// TwinCAT 3 PLC project BMS_Allerstorfer
// ProgramVersion: 3.1.4024.0
// libraries:
//   EfficientIO Communicator, * (EfficientIO)
//   EfficientIO ModbusTCP, * (EfficientIO)
//   Lynus Energy Basic, * (Lynus AG)
//   Lynus Persistent Data V1, * (Lynus AG)
//   Lynus Standards, * (Lynus AG)
//   Tc2_IoFunctions, * (Beckhoff Automation GmbH)
//   Tc2_ModbusSrv, * (Beckhoff Automation GmbH)
//   Tc2_Standard, * (Beckhoff Automation GmbH)
//   Tc2_System, * (Beckhoff Automation GmbH)
//   Tc2_Utilities, * (Beckhoff Automation GmbH)
//   Tc3_BA_Common, * (Beckhoff Automation GmbH)
//   Tc3_Module, * (Beckhoff Automation GmbH)
// project tree:
//   / FastTask.TcTTO, MiddleTask.TcTTO, SlowTask.TcTTO
//   FB/ FB_3HeaterControl.TcPOU, FB_HourCounter.TcPOU, FB_LinearEquation.TcPOU (not stored), FB_PID_T.TcPOU (not stored), FB_RAMP.TcPOU, FB_Symo_PV_Inverter_FLOAT_1_DM_30_InclDisable.TcPOU (not stored), FB_Symo_PV_Inverter_FLOAT_1_DM_30_InclDisable_original.TcPOU
//   POUs/ prgComEffIO.TcPOU, prgEMS.TcPOU, prgGrid.TcPOU, prgHouse.TcPOU, prgPersistent.TcPOU, prgPV.TcPOU, prgRWEffIO.TcPOU (not stored), prgTemperature.TcPOU, prgVarEffIO.TcPOU
// real-time tasks:
//   TASK PlcTask1: cycle T#10ms, priority 21, ADS port 351
//   TASK PlcTask: cycle T#10ms, priority 20, ADS port 350
//   TASK SlowTask: cycle T#10ms, priority 22, ADS port 352
// I/O:
//   DEVICE Gerät 2 (CX-BK)
//     Box 1 (CX-BK)
// variable links:
//   BMS_Allerstorfer/BMS_Allerstorfer Instance <-> Device 2 (CX-BK)/Box 1 (CX-BK)
//     MiddleTask Inputs/prgGrid.fbEM1.fbKL3403.byStateCH1 <-> Term 5 (KL3403)/Channel 1/Status
//     MiddleTask Inputs/prgGrid.fbEM1.fbKL3403.byStateCH2 <-> Term 5 (KL3403)/Channel 2/Status
//     MiddleTask Inputs/prgGrid.fbEM1.fbKL3403.byStateCH3 <-> Term 5 (KL3403)/Channel 3/Status
//     MiddleTask Inputs/prgGrid.fbEM1.fbKL3403.iDataInCH1 <-> Term 5 (KL3403)/Channel 1/Daten Ein
//     MiddleTask Inputs/prgGrid.fbEM1.fbKL3403.iDataInCH2 <-> Term 5 (KL3403)/Channel 2/Daten Ein
//     MiddleTask Inputs/prgGrid.fbEM1.fbKL3403.iDataInCH3 <-> Term 5 (KL3403)/Channel 3/Daten Ein
//     MiddleTask Inputs/prgGrid.fbKBusState.uiKBusState_OUT <-> Inputs/State
//     MiddleTask Inputs/prgTemperature.stInData_{1..4}/iDataIn <-> Term 4 (KL3204)/Channel {1..4}/Daten Ein  (4 links)
//     MiddleTask Inputs/prgTemperature.stInData_{1..4}/iState <-> Term 4 (KL3204)/Channel {1..4}/Status  (4 links)
//     MiddleTask Outputs/prgGrid.fbEM1.fbKL3403.byCntrCH1 <-> Term 5 (KL3403)/Channel 1/Kontrolle
//     MiddleTask Outputs/prgGrid.fbEM1.fbKL3403.byCntrCH2 <-> Term 5 (KL3403)/Channel 2/Kontrolle
//     MiddleTask Outputs/prgGrid.fbEM1.fbKL3403.byCntrCH3 <-> Term 5 (KL3403)/Channel 3/Kontrolle
//     MiddleTask Outputs/prgTemperature.mOut_1 <-> Term 3 (KL2408)/Channel 1/Ausgang
//     MiddleTask Outputs/prgTemperature.mOut_2 <-> Term 3 (KL2408)/Channel 2/Ausgang
//     MiddleTask Outputs/prgTemperature.mOut_3 <-> Term 3 (KL2408)/Channel 3/Ausgang
//     MiddleTask Outputs/prgTemperature.stOutData_{1..4}/iCtrl <-> Term 4 (KL3204)/Channel {1..4}/Kontrolle  (4 links)
//     MiddleTask Outputs/prgTemperature.stOutData_{1..4}/iDataOut <-> Term 4 (KL3204)/Channel {1..4}/Daten Aus  (4 links)
//     SlowTask Outputs/prgTemperature.mOut_{4..8} <-> Term 3 (KL2408)/Channel {4..8}/Ausgang  (5 links)

CONFIGURATION BMS_Allerstorfer
    RESOURCE PLC ON TwinCAT3
        TASK FastTask(INTERVAL := T#10ms, PRIORITY := 21);
        TASK MiddleTask(INTERVAL := T#10ms, PRIORITY := 20);
        TASK SlowTask(INTERVAL := T#10ms, PRIORITY := 22);
        PROGRAM prgVarEffIO WITH FastTask : prgVarEffIO;
        PROGRAM prgRWEffIO WITH FastTask : prgRWEffIO;
        PROGRAM prgComEffIO WITH MiddleTask : prgComEffIO;
        PROGRAM prgEMS WITH MiddleTask : prgEMS;
        PROGRAM prgGrid WITH MiddleTask : prgGrid;
        PROGRAM prgHouse WITH MiddleTask : prgHouse;
        PROGRAM prgPersistent WITH MiddleTask : prgPersistent;
        PROGRAM prgTemperature WITH MiddleTask : prgTemperature;
        PROGRAM prgPV WITH MiddleTask : prgPV;
        PROGRAM prgComEffIO WITH SlowTask : prgComEffIO;
    END_RESOURCE
END_CONFIGURATION

// ---- POUs/prgVarEffIO.TcPOU
PROGRAM prgVarEffIO
VAR
	fbVar		: FB_VarInfo_V3;
END_VAR

fbVar(
	bReadInfo:= , 
	eTMCFile:= eSelectTMCFile.eDontUseTMCFile, 
	eSavePositionTMCFile:= eSavePositionOnPLC.ePostionHardDisk, 
	udiCounterFoundVariables=> , 
	bError=> , 
	bBusy=> , 
	byProgress=> , 
	udiErrorCodeOut=> , 
	eErrorVarInfo_Out=> , 
	sVarWithError=> );
	
fbVar(
	bReadInfo:= , 
	eTMCFile:= eSelectTMCFile.eDontUseTMCFile, 
	eSavePositionTMCFile:= eSavePositionOnPLC.ePostionHardDisk, 
	udiCounterFoundVariables=> , 
	bError=> , 
	bBusy=> , 
	byProgress=> , 
	udiErrorCodeOut=> , 
	eErrorVarInfo_Out=> , 
	sVarWithError=> );
	
fbVar(
	bReadInfo:= , 
	eTMCFile:= eSelectTMCFile.eDontUseTMCFile, 
	eSavePositionTMCFile:= eSavePositionOnPLC.ePostionHardDisk, 
	udiCounterFoundVariables=> , 
	bError=> , 
	bBusy=> , 
	byProgress=> , 
	udiErrorCodeOut=> , 
	eErrorVarInfo_Out=> , 
	sVarWithError=> );

END_PROGRAM

// ---- POUs/prgComEffIO.TcPOU
PROGRAM prgComEffIO
VAR
	fbCom		: FB_MqttCommunicator_V3;
	strAuthKey: STRING(INT#14);
END_VAR

fbCom(
	bConnect:= TRUE, 
	strAuthKey:= 'BMS99299754422', 
	sUserName:= '23fb7b57-8617-4e5d-874b-d9d19721e991', 					// adopt MQTT Username
	sUserPassword:= '60c350ff-dfc0-4bd2-861d-a7d102b328dc', 				// adopt MQTT Password
	eSavePositionCertificate:= eSavePositionOnPLC.ePostionHardDisk, 
	bConnected=> , 
	bError=> , 
	hrErrorCode=> , 
	eConnectionState=> , 
	eErrorMessage_Out=> );
	
	(* old
		strAuthKey:= 'EIO08031879806', 
	sUserName:= 'b37f3835-35ae-441a-9870-02e312a14f46', 					// adopt MQTT Username
	sUserPassword:= '800bfb28-4995-4679-af93-39628385cccf', 				// adopt MQTT Password
*)

END_PROGRAM

// ---- POUs/prgEMS.TcPOU
PROGRAM prgEMS
VAR PERSISTENT
	byMaxDepthOfDischrgEPO		: BYTE;							//{#lynus.ag#()}
	byPrioMinChrgBattSOCInEPO	: BYTE;							//{#lynus.ag#()}
	byResChrgfromGridToBatt		: BYTE;							//{#lynus.ag#()}
	byReserveSOCEPO				: BYTE;							//{#lynus.ag#()}
	uiUpdateTime				: UINT;							//{#lynus.ag#()}
	bEnableEMS					: BOOL;							//{#lynus.ag#()}
	bAllowChrgFromGrid			: BOOL;							//{#lynus.ag#()}
	rMainFuseCSEMS				: REAL;							//{#lynus.ag#()}
	iOperationModeEMS			: INT;							//{#lynus.ag#()}
END_VAR
VAR
	fbEMS						: FB_EMS;
	bIsEnableEMS				: BOOL;							//{#lynus.ag#()}
	bStateAllowChrgFromGrid		: BOOL;							//{#lynus.ag#()}
	bHPActivate					: BOOL;							//{#lynus.ag#()}
	bControllingState			: BOOL;							//{#lynus.ag#()}
	iMessageEMS					: INT;							//{#lynus.ag#()}
	rHeartbeatEMS				: REAL;							//{#lynus.ag#()}
	rErrorWarningEMS			: REAL;							//{#lynus.ag#()}
	rReadyEMS					: REAL;							//{#lynus.ag#()}
	rNewBatteryPowerEMS			: REAL;							//{#lynus.ag#()}
END_VAR

fbEMS.stSetupEMS.bAllowChrgFromGrid := bAllowChrgFromGrid;
	fbEMS.stSetupEMS.byMaxDepthOfDischrgEPO := byMaxDepthOfDischrgEPO;
		fbEMS.stSetupEMS.byPrioMinChrgBattSOCInEPO := byPrioMinChrgBattSOCInEPO;
			fbEMS.stSetupEMS.byResChrgfromGridToBatt := byResChrgfromGridToBatt;
				fbEMS.stSetupEMS.byReserveSOCEPO := byReserveSOCEPO;
					fbEMS.stSetupEMS.rSizeMainFuseCS := rMainFuseCSEMS;
						fbEMS.stSetupEMS.uiUpdateTime := uiUpdateTime;

IF iOperationModeEMS = 0 THEN fbEMS.eOperationMode := E_OperatingMode_EMS.eAllOff;
ELSIF iOperationModeEMS = 1 THEN fbEMS.eOperationMode := E_OperatingMode_EMS.eSelfConsumption;	
ELSIF iOperationModeEMS = 2 THEN fbEMS.eOperationMode := E_OperatingMode_EMS.ePeakLoadCapping;
ELSIF iOperationModeEMS = 3 THEN fbEMS.eOperationMode := E_OperatingMode_EMS.eLoadManagement;			
END_IF

fbEMS(
	bEnable:= bEnableEMS, 
	diNrOfEM_IN_ECS:= , 
	stSetupEMS:= , 
	eOperationMode:= , 
	eSpeedModeBackendController:= E_SpeedModeBackendController_EMS.eSlow, 
	eSpeedModeLocalController:= E_SpeedModeLocalController_EMS.eSlow,
	bActivateHP:= bHPActivate, 
	bControllingState:= TRUE, // bControllingState, 
	rHeartbeat:= rHeartbeatEMS, 
	rErrorWarning:= rErrorWarningEMS, 
	rEnergyOptReady:= rReadyEMS, 
	rNewBattPower:= rNewBatteryPowerEMS, 
	eMessageEMS=> iMessageEMS, 
	bStateEnable=> bIsEnableEMS, 
	bStateAllowChrgFromGrid=> bStateAllowChrgFromGrid, 
	bMissingPowerData=> , 
	bSurplusAvailable=> , 
	byProgress=> , 
	uiState_OUT=> , 
	diNrOfEMS_OUT=> , 
	arrMinPrioReached=> , 
	arrMaxPrioReached=> );

END_PROGRAM

// ---- POUs/prgGrid.TcPOU
PROGRAM prgGrid
VAR PERSISTENT
	rSizeGridConn				: REAL;									//{#lynus.ag#()}
	lrCounterGridCon			: LREAL;							//{#lynus.ag#()}
	lrCounterGridProd			: LREAL;							//{#lynus.ag#()}

END_VAR
VAR
	fbKBusState					: FB_K_Bus_State;
	fbEM1						: FB_EM_Beckhoff_KL3403;
	fbGrid						: FB_Grid_Power;
	fbGridCounter				: FB_EnergyCounter;
	lrPowerGrid					: LREAL;							//{#lynus.ag#()}
	lrPowerEM1_1				: LREAL;							//{#lynus.ag#()}
	lrPowerEM1_2				: LREAL;							//{#lynus.ag#()}
	lrPowerEM1_3				: LREAL;							//{#lynus.ag#()}
	lr_GridVoltageL1N_V			: LREAL;							//{#lynus.ag#()}
	lr_GridVoltageL2N_V			: LREAL;							//{#lynus.ag#()}
	lr_GridVoltageL3N_V			: LREAL;							//{#lynus.ag#()}

	lrReactivePowerGrid			: LREAL;							//{#lynus.ag#()}
	lrApparentPowerGrid			: LREAL;							//{#lynus.ag#()}
	lrPowerGridCons				: LREAL;							//{#lynus.ag#()}
	lrPowerGridProd				: LREAL;							//{#lynus.ag#()}
END_VAR

fbKBusState(	uiKBusState_OUT=> , 
				b_Kbus_notOk=> , 
				word_ErrorCount=> );


fbEM1(
	bEnable:= TRUE, 
	bChannel1Invers:= FALSE,				//Invert power data when transformer are mounted upside down
	bChannel2Invers:= FALSE, 
	bChannel3Invers:= false, 
	uiCurrentTransformerRatioL1:= 250, // 250 / 5 A CTs mounted
	uiCurrentTransformerRatioL2:= 250, 
	uiCurrentTransformerRatioL3:= 250, 
	uiKBusState_IN:= fbKBusState.uiKBusState_OUT, 
	stDataEMPower=> , 
	stDataEMCounter=> , 
	stDataEMPowerRealTime=> , 
	stDataEMCounterRealTime=> , 
	diNrOfEM_OUT=> );

lrPowerGrid := fbEM1.stDataEMPower.lrPowerTotal;
lrCounterGridCon := fbEM1.stDataEMCounter.lrTotalCounterEnergy_Consumption;	
lrCounterGridProd := fbEM1.stDataEMCounter.lrTotalCounterEnergy_Production;	
lrPowerEM1_1 := fbEM1.stDataEMPower.lrPowerL1;
lrPowerEM1_2 := fbEM1.stDataEMPower.lrPowerL2;
lrPowerEM1_3 := fbEM1.stDataEMPower.lrPowerL3;

lrReactivePowerGrid:=fbEM1.stDataEMPower.lrReactivePowerTotal;
lrApparentPowerGrid:=fbEM1.stDataEMPower.lrApparentPowerTotal;

lr_GridVoltageL1N_V:=fbEM1.stDataEMPower.lrVoltageL1N;
lr_GridVoltageL2N_V:=fbEM1.stDataEMPower.lrVoltageL2N;
lr_GridVoltageL3N_V:=fbEM1.stDataEMPower.lrVoltageL3N;


fbGrid(
	bEnable:= TRUE, 
	diNrOfEMS_IN:= prgEMS.fbEMS.diNrOfEMS_OUT, 
	diNrOfEM_IN_Grid:= fbEM1.diNrOfEM_OUT, 
	rSizeGridConn:= rSizeGridConn, 
	stDataGrid=> , 
	diNrOfGrid_OUT=> );
	



// EnergyCounter
fbGridCounter(
	byActiveTariff:= 1, 
	lrPowerInput:= lrPowerGrid, 
	lrTotalCounterEnergy_Consumption=> , 
	lrTotalCounterEnergy_Production=> , 
	lrCounterEnergyT1_Consumption=> , 
	lrCounterEnergyT2_Consumption=> , 
	lrCounterEnergyT1_Production=> , 
	lrCounterEnergyT2_Production=> );

IF fbGridCounter.lrTotalCounterEnergy_Production > lrCounterGridProd THEN  	
		lrCounterGridProd := fbGridCounter.lrTotalCounterEnergy_Production;
END_IF

IF fbGridCounter.lrTotalCounterEnergy_Consumption > lrCounterGridCon THEN  	
	lrCounterGridCon := fbGridCounter.lrTotalCounterEnergy_Consumption;
END_IF

lrPowerGridCons := fbEM1.stDataEMPower.lrPowerConsumption;
lrPowerGridProd := fbEM1.stDataEMPower.lrPowerProduction;

END_PROGRAM

// ---- POUs/prgHouse.TcPOU
PROGRAM prgHouse
VAR
	fbHouse				: FB_HouseC_Power_Virtual;
	bHouseEnabled		: BOOL;						//{#lynus.ag#()}
	lrPowerHouse		: LREAL;					//{#lynus.ag#()}
	lrPowerHouse_Manual	: LREAL;					//{#lynus.ag#()}
	lrPowerHouseUndelayed: LREAL;					//{#lynus.ag#()}
END_VAR
VAR PERSISTENT
	bEnableHouse		: BOOL;						//{#lynus.ag#()}
END_VAR

fbHouse(
	bEnable:= bEnableHouse, 
	diNrOfEMS_IN:= prgEMS.fbEMS.diNrOfEMS_OUT, 
	bSetDefault:= , 
	lrCounterConsumptionSetDefault:= , 
	lrCounterProductionSetDefault:= , 
	stDataHouseC=> , 
	diNrOfHouseC_OUT=> );
	
bHouseEnabled := fbHouse.stDataHouseC.bEnabled;
// lrPowerHouse := fbHouse.stDataHouseC.lrPower; 		// not calculating correctly	
lrPowerHouse_Manual := prgPV.lrPowerPV + prgGrid.lrPowerGrid;

lrPowerHouse:= MAX(0,lrPowerHouse_Manual)- prgTemperature.real_PowerHeater;
lrPowerHouseUndelayed := prgGrid.fbEM1.stDataEMPowerRealTime.lrPowerTotal + prgPV.lrPowerPV - prgTemperature.real_PowerHeater;

END_PROGRAM

// ---- POUs/prgPV.TcPOU
PROGRAM prgPV
VAR PERSISTENT
	lrCounterPV				: LREAL;									//{#lynus.ag#()}
	str_IP_PV_1				: STRING(15):= '10.11.90.100';
	arr_b_EnableWrite			: ARRAY[1..30] OF BOOL;								// Enable write function
	arr_m_DisableInverter		: ARRAY[1..30] OF BOOL;								// disable inverter 
	arr_int_InverterSetpoint	: ARRAY[1..30] OF INT;								// inverter setpoint i[1/100 %] 
	real_MainsSetpointRegulate	: REAL:=-20;							//{#lynus.ag#()}
	real_Factor_Calc: REAL:=110;
	rPValue: REAL := 2;
	udint_IValue: UDINT:=250;
	uditn_DValue: UDINT:=30;
	realMaxGridPower_1: REAL:=-35;
	realMaxGridPower_2: REAL:=-40;
END_VAR
VAR
	fbPV_1					: FB_Symo_PV_Inverter_FLOAT_1_DM_30_InclDisable;
	fbPVCounter				: FB_EnergyCounter;
	lrPowerPV				: LREAL;				//{#lynus.ag#()}
	byErrorWarningPV		: BYTE;					//{#lynus.ag#()}
	
	// extend or reduce amount of PV Inverters
	lrPowerPV_1				: LREAL;				//{#lynus.ag#()}
	lrPowerPV_2				: LREAL;				//{#lynus.ag#()}

	int_SetPointInverter	:INT;					//{#lynus.ag#()}

	real_ActualLoadPercent_PV1: REAL;				//{#lynus.ag#()}
	real_ActualLoadPercent_PV2: REAL;				//{#lynus.ag#()}
	real_RegulatroMaxValue_Calc: REAL;				//{#lynus.ag#()}
	FB_PID_Inverter :FB_PID_T;
	ton_PV_On_Delay_after_Off :ARRAY[1..2]OF Ton;
	
	real_Setpoint_PID_In: REAL;					//{#lynus.ag#()}
	real_RegulatroMaxValue_Limit: REAL;				//{#lynus.ag#()}
		
	i: INT;
END_VAR

// write setpoints to PV array
arr_int_InverterSetpoint[1] := int_SetPointInverter;
arr_int_InverterSetpoint[2] := int_SetPointInverter;

// limit mains regulator setpoint
real_MainsSetpointRegulate := LIMIT(-30,real_MainsSetpointRegulate,0); 
 

fbPV_1.arrUnitID_Inverter[1]:=1;
fbPV_1.arr_b_EnableWrite[1] := arr_b_EnableWrite[1];
fbPV_1.arr_m_DisableInverter[1] := arr_m_DisableInverter[1];
fbPV_1.arr_int_InverterSetpoint[1] := arr_int_InverterSetpoint[1];

fbPV_1.arrUnitID_Inverter[2]:=2;
fbPV_1.arr_b_EnableWrite[2] := arr_b_EnableWrite[2];
fbPV_1.arr_m_DisableInverter[2] := arr_m_DisableInverter[2];
fbPV_1.arr_int_InverterSetpoint[2] := arr_int_InverterSetpoint[2];


fbPV_1.arrUnitID_Inverter[1] :=1;
fbPV_1(
	bEnable				:= TRUE, 
	sIPAdress			:= str_IP_PV_1, 			// modify IP Adress
	arrUnitID_Inverter	:= ,
	arr_b_EnableWrite	:=,
	arr_m_DisableInverter := ,
	arrDataSymo10		=> ,
	stDataEMPower_PV	=> , 
	stDataEMCounter_PV	=> , 
	diNrOfEM_OUT_PV		=> );

lrPowerPV_1 := fbPV_1.arrDataSymo10[1].lrPowerAcInverter;
lrPowerPV_2 := fbPV_1.arrDataSymo10[2].lrPowerAcInverter;




lrPowerPV := lrPowerPV_1 + lrPowerPV_2 ;

// EnergyCounter
fbPVCounter(
	byActiveTariff:= 1, 
	lrPowerInput:= 0 - lrPowerPV, 
	lrTotalCounterEnergy_Consumption=> , 
	lrTotalCounterEnergy_Production=> , 
	lrCounterEnergyT1_Consumption=> , 
	lrCounterEnergyT2_Consumption=> , 
	lrCounterEnergyT1_Production=> , 
	lrCounterEnergyT2_Production=> );
	
IF fbPVCounter.lrTotalCounterEnergy_Production > lrCounterPV THEN  	
	lrCounterPV := fbPVCounter.lrTotalCounterEnergy_Production;
END_IF

// calculate maximum regulator value by looking at the nomal inverter power 
// nominal inverter Values	PV1: 27kW / PV2: 27kW 
real_ActualLoadPercent_PV1 := LREAL_TO_REAL(lrPowerPV_1) / 27*100;
real_ActualLoadPercent_PV2 := LREAL_TO_REAL(lrPowerPV_2) / 27*100;

real_RegulatroMaxValue_Calc := 	MAX(real_ActualLoadPercent_PV1,real_ActualLoadPercent_PV2);
real_RegulatroMaxValue_Calc := LIMIT(1,real_RegulatroMaxValue_Calc,100);
real_RegulatroMaxValue_Limit := LIMIT(0,real_RegulatroMaxValue_Calc*real_Factor_Calc,10000);	// add 20% regualtion margin
FB_PID_Inverter.rMaxValue := real_RegulatroMaxValue_Limit;

// mains parallel operation

FB_PID_Inverter.bEnable := TRUE;
FB_PID_Inverter.rSetpoint := LREAL_TO_REAL(- real_MainsSetpointRegulate); 
int_SetPointInverter := REAL_TO_INT(FB_PID_Inverter.rQController);
FB_PID_Inverter.rActualValue:= LREAL_TO_REAL( -prgGrid.fbEM1.stDataEMPowerRealTime.lrPowerTotal);


FB_PID_Inverter(
	bEnable:= , 
	rSetpoint:= , 
	udiIValue:= udint_IValue, 
	udiDValue:= uditn_DValue, 
	udiDamping:= 0, 
	rPValue:= rPValue, 
	rMaxValue:= , 
	rMinValue:= 100, 
	rNeutralZone:= 1, 
	bDirection:= FALSE, 
	rActualValue:= ,
	rQController=> );
	

real_Setpoint_PID_In := FB_PID_Inverter.rSetpoint;



// disable inverters in case of mains power too big
IF prgGrid.fbEM1.stDataEMPowerRealTime.lrPowerTotal < realMaxGridPower_1 THEN
	arr_m_DisableInverter[1] := TRUE;
ELSIF prgGrid.fbEM1.stDataEMPowerRealTime.lrPowerTotal < realMaxGridPower_2 THEN
	arr_m_DisableInverter[2] := TRUE;
END_IF
IF prgGrid.fbEM1.stDataEMPowerRealTime.lrPowerTotal < -50 THEN
	arr_m_DisableInverter[1] := TRUE;
	arr_m_DisableInverter[2] := TRUE;
END_IF
FOR i:= 1 TO 2 BY 1 DO
	IF arr_m_DisableInverter[i] = TRUE THEN
		ton_PV_On_Delay_after_Off[i].IN := TRUE;
	END_IF
	IF ton_PV_On_Delay_after_Off[i].Q THEN
		ton_PV_On_Delay_after_Off[i].IN := FALSE;
		arr_m_DisableInverter[i] := FALSE;
	END_IF
		
END_FOR
ton_PV_On_Delay_after_Off[1]( PT := T#30S); 	
ton_PV_On_Delay_after_Off[2]( PT := T#60S);

END_PROGRAM

// ---- POUs/prgTemperature.TcPOU
PROGRAM prgTemperature
VAR
	
	fb_Config			: FB_KL320xConfig;
	stInData_1   AT%I*		: ST_KL320xInData;
	stOutData_1  AT%Q*		: ST_KL320xOutData;
	stInData_2   AT%I*		: ST_KL320xInData;
	stOutData_2  AT%Q*		: ST_KL320xOutData;
	stInData_3   AT%I*		: ST_KL320xInData;
	stOutData_3  AT%Q*		: ST_KL320xOutData;
	stInData_4   AT%I*		: ST_KL320xInData;
	stOutData_4  AT%Q*		: ST_KL320xOutData;
	stInData_temp	: ST_KL320xInData;
	stOutData_temp	: ST_KL320xOutData;

	x: INT;
	real_Temp_BoilerOben	:REAL;				//{#lynus.ag#()}
	real_Temp_BoilerUnten	:REAL;				//{#lynus.ag#()}
	mOut_1  AT%Q*		: BOOL;
	mOut_2  AT%Q*		: BOOL;
	mOut_3  AT%Q*		: BOOL;
	mOut_4  AT%Q*		: BOOL;
	mOut_5  AT%Q*		: BOOL;
	mOut_6  AT%Q*		: BOOL;
	mOut_7  AT%Q*		: BOOL;
	mOut_8  AT%Q*		: BOOL;
	fb_heater:FB_3HeaterControl;

	b_Heater1_On: BOOL;							//{#lynus.ag#()}
	b_Heater2_On: BOOL;							//{#lynus.ag#()}
	b_Heater3_On: BOOL;							//{#lynus.ag#()}
	b_Heater1_Manual_On: BOOL;							//{#lynus.ag#()}
	b_Heater2_Manual_On: BOOL;							//{#lynus.ag#()}
	b_Heater3_Manual_On: BOOL;							//{#lynus.ag#()}
	real_StepHeaterControl	: REAL;				//{#lynus.ag#()}
	real_PowerHeater1		: REAL;				//{#lynus.ag#()}
	real_PowerHeater2		: REAL;				//{#lynus.ag#()}
	real_PowerHeater3		: REAL;				//{#lynus.ag#()}
	real_PowerHeater		: REAL;				//{#lynus.ag#()}
END_VAR
VAR PERSISTENT
	real_Boiler_SetPoint	: REAL:=70;				//{#lynus.ag#()}
	b_Enable				: BOOL;					//{#lynus.ag#()}

END_VAR




real_Temp_BoilerUnten :=  INT_TO_REAL(stInData_1.iDataIn)/10;
real_Temp_BoilerOben  :=  INT_TO_REAL(stInData_2.iDataIn)/10;

// heater control
fb_heater(
	m_Enbale:= b_Enable , 
	m_Temperature_high:=  MAX(real_Temp_BoilerOben,real_Temp_BoilerUnten)>95, 
	m_Battery_Discharging := FALSE,
	real_Temperature:=  MAX(real_Temp_BoilerOben,real_Temp_BoilerUnten), 
	real_TemperatureSetPoint:= real_Boiler_SetPoint, 
	real_GridPower := LREAL_TO_REAL(prgGrid.lrPowerGrid), 
	real_BatteryPower := 0,
	real_Size_Step1_kW:= 6, 
	real_Size_Step2_kW:= 6, 
	real_Size_Step3_kW:= 6, 
	m_Step1=> b_Heater1_On, 
	m_Step2=> b_Heater2_On, 
	m_Step3=> b_Heater3_On);
	
mOut_1 := 	b_Heater1_On OR b_Heater1_Manual_On;
mOut_2 := 	b_Heater2_On OR b_Heater2_Manual_On;
mOut_3 := 	b_Heater3_On or b_Heater3_Manual_On;


IF mOut_1 THEN
	real_PowerHeater1 := fb_heater.real_Size_Step1_kW;
ELSE
	real_PowerHeater1 := 0;
END_IF
IF mOut_2 THEN
	real_PowerHeater2 := fb_heater.real_Size_Step2_kW;
ELSE
	real_PowerHeater2 := 0;
END_IF
IF mOut_3 THEN
	real_PowerHeater3 := fb_heater.real_Size_Step3_kW;
ELSE
	real_PowerHeater3 := 0;
END_IF
real_StepHeaterControl := SINT_TO_REAL(fb_heater.sint_Steps_On);

real_PowerHeater := real_PowerHeater1 + real_PowerHeater2 + real_PowerHeater3;
	
CASE x OF 
	0:
		fb_Config.bConfigurate := FALSE;
	1:
		stInData_temp  := stInData_1;
		stOutData_1 	:=stOutData_temp ;
	2:
		stInData_temp  := stInData_2;
		stOutData_2 	:=stOutData_temp ;
	3:
		stInData_temp  := stInData_3;
		stOutData_3 	:=stOutData_temp ;
	4:
		stInData_temp  := stInData_4;
		stOutData_4 	:=stOutData_temp ;
	
END_CASE
// set iSetSensorType = 2 for PT1000
fb_Config(
	bConfigurate:= , 
	bReadConfig:= , 
	iSetSensorType:= , 
	tTimeout:= , 
	bBusy=> , 
	bError=> , 
	iErrorId=> , 
	iState=> , 
	iDataIn=> , 
	iTerminalType=> , 
	iSpecialType=> , 
	iFirmwareVersion=> , 
	sDescription=> , 
	sSensorType=> , 
	bTwoWiredConnection=> , 
	stInData:= stInData_temp , 
	stOutData:= stOutData_temp);

END_PROGRAM

// ---- FB/FB_3HeaterControl.TcPOU
FUNCTION_BLOCK FB_3HeaterControl
VAR_INPUT
	m_Enbale					: BOOL;
	m_Temperature_high			: BOOL;
	m_Battery_Discharging		: BOOL;
	real_Temperature			: REAL;
	real_TemperatureSetPoint	: REAL;
	real_GridPower				: REAL;
	real_BatteryPower			: REAL;
	real_Size_Step1_kW			: REAL;
	real_Size_Step2_kW			: REAL;
	real_Size_Step3_kW			: REAL;
	
	
END_VAR
VAR_OUTPUT
	m_Step1						: BOOL;
	m_Step2						: BOOL;
	m_Step3						: BOOL;
END_VAR
VAR
	fb_HourCounter_Step1		: FB_HourCounter;
	fb_HourCounter_Step2		: FB_HourCounter;
	fb_HourCounter_Step3		: FB_HourCounter;
	r_Trig_allOff				: r_trig;
	real_Hours_Step1			: REAL;
	real_Hours_Step2			: REAL;
	real_Hours_Step3			: REAL;	
	arr_sint_StartOrder			: ARRAY[1..3] OF SINT;
	arr_real_LoadSize			: ARRAY[1..3] OF REAL;
	arr_real_Steps				: ARRAY[1..3] OF REAL;
	
	
	int_state					: INT;
	ton_OnDelay_Steps			: Ton;
	time_OnDelay				: TIME:=T#30S;	
	ton_OffDelay_Steps			: Ton;
	time_OffDelay				: TIME:=T#30S;	
	ton_WaitDelay_Steps			: Ton;
	time_WaitDelay				: TIME:=T#30S;	
	sint_Steps_On				: SINT;
	ton_OffDelay2_Steps			: Ton;
	time_OffDelay2				: TIME:=T#15S;	
END_VAR


CASE int_state OF
	0:	// not enabled
		m_Step1 := FALSE;
		m_Step2 := FALSE;
		m_Step3 := FALSE;
		sint_Steps_On := 0;
		ton_OnDelay_Steps.IN := FALSE;
		ton_OffDelay_Steps.IN := FALSE;
		ton_OffDelay2_Steps.IN := FALSE;
		ton_WaitDelay_Steps.IN := FALSE;
		
		IF 	m_Enbale THEN
			int_state := 10;
		END_IF
	
	10: // check that mains power gets more negative thenn step power + 20%
		IF sint_Steps_On <3 THEN 
			IF real_GridPower + arr_real_LoadSize[sint_Steps_On+1]*1.2 < 0 AND NOT m_Temperature_high AND real_Temperature < (real_TemperatureSetPoint-2) THEN 
				ton_OnDelay_Steps.IN := TRUE;
			ELSE
				ton_OnDelay_Steps.IN := FALSE;
			END_IF
		END_IF
		IF ton_OnDelay_Steps.Q THEN
			ton_OnDelay_Steps.IN := FALSE;
			int_state := 11;
		END_IF
		IF sint_Steps_On <>0 THEN 
			IF real_GridPower > 3 OR  real_Temperature > real_TemperatureSetPoint OR (m_Battery_Discharging AND real_BatteryPower > 5) THEN
 				ton_OffDelay_Steps.IN := TRUE;
			ELSE
				ton_OffDelay_Steps.IN := FALSE;
			END_IF
			IF real_GridPower > 10 THEN
 				ton_OffDelay2_Steps.IN := TRUE;
			ELSE
				ton_OffDelay2_Steps.IN := FALSE;
			END_IF
			
			IF ton_OffDelay_Steps.Q THEN
				ton_OffDelay_Steps.IN := FALSE;
				ton_OffDelay2_Steps.IN := FALSE;
				int_state := 12;
			END_IF
			IF m_Temperature_high AND sint_Steps_On <>0 THEN
				ton_OnDelay_Steps.IN := FALSE;
 				ton_OffDelay_Steps.IN := FALSE;
				ton_OffDelay2_Steps.IN := FALSE;
				int_state := 15;
			END_IF
		END_IF
		
		
	11: // count step one up
		sint_Steps_On := sint_Steps_On+1;
		int_state := 20;
		
	12:// count step one down
		sint_Steps_On := sint_Steps_On-1;
		int_state := 20;
	
	15:// Switch off all steps
		sint_Steps_On := 0;
		int_state := 20;
	
	20: // wait state	
		ton_WaitDelay_Steps.IN := TRUE;
		IF ton_WaitDelay_Steps.Q THEN
			ton_WaitDelay_Steps.IN := FALSE;
			int_state := 10;
		END_IF
END_CASE
ton_OnDelay_Steps(PT := time_OnDelay);
ton_OffDelay_Steps(PT := time_OffDelay);
ton_OffDelay2_Steps(PT := time_OffDelay2);
ton_WaitDelay_Steps(PT := time_WaitDelay);

// if not enabled, force state to 0
IF 	NOT m_Enbale THEN
	int_state := 0;
END_IF

// switch on steps according to sint_Steps_On
CASE sint_Steps_On OF
	0:
		m_Step1 := FALSE;
		m_Step2 := FALSE;
		m_Step3 := FALSE;
		
	1:
		m_Step1 := FALSE;
		m_Step2 := FALSE;
		m_Step3 := FALSE;
		IF arr_sint_StartOrder[1] = 1 THEN 
 			m_Step1 := TRUE;
		ELSIF arr_sint_StartOrder[1] = 2 THEN 
			m_Step2 := TRUE;
		ELSIF arr_sint_StartOrder[1] = 3 THEN 
			m_Step3 := TRUE;
		END_IF
	2:
		m_Step1 := FALSE;
		m_Step2 := FALSE;
		m_Step3 := FALSE;
		IF arr_sint_StartOrder[1] = 1 THEN 
 			m_Step1 := TRUE;
		ELSIF arr_sint_StartOrder[1] = 2 THEN 
			m_Step2 := TRUE;
		ELSIF arr_sint_StartOrder[1] = 3 THEN 
			m_Step3 := TRUE;
		END_IF
		IF arr_sint_StartOrder[2] = 1 THEN 
 			m_Step1 := TRUE;
		ELSIF arr_sint_StartOrder[2] = 2 THEN 
			m_Step2 := TRUE;
		ELSIF arr_sint_StartOrder[2] = 3 THEN 
			m_Step3 := TRUE;
		END_IF
	3:
		m_Step1 := TRUE;
		m_Step2 := TRUE;
		m_Step3 := TRUE;		
END_CASE		
	
// find out which step has the lowest running hours
r_Trig_allOff(CLK := NOT m_Step1 AND NOT m_Step2 AND NOT m_Step3);

IF r_Trig_allOff.Q THEN
	IF real_Hours_Step1 <= real_Hours_Step2 AND real_Hours_Step1<=real_Hours_Step3 THEN
		arr_sint_StartOrder[1] := 1;
		IF real_Hours_Step2 <= real_Hours_Step3 THEN
			arr_sint_StartOrder[2] := 2;
			arr_sint_StartOrder[3] := 3;
		ELSE
			arr_sint_StartOrder[2] := 3;
			arr_sint_StartOrder[3] := 2;
		END_IF
	ELSIF real_Hours_Step2 <= real_Hours_Step1 AND real_Hours_Step2<=real_Hours_Step3 THEN
		arr_sint_StartOrder[1] := 2;
		IF real_Hours_Step1 <= real_Hours_Step3 THEN
			arr_sint_StartOrder[2] := 1;
			arr_sint_StartOrder[3] := 3;
		ELSE
			arr_sint_StartOrder[2] := 3;
			arr_sint_StartOrder[3] := 1;
		END_IF
	ELSIF real_Hours_Step3 <= real_Hours_Step1 AND real_Hours_Step3<=real_Hours_Step2 THEN
		arr_sint_StartOrder[1] := 3;
		IF real_Hours_Step1 <= real_Hours_Step2 THEN
			arr_sint_StartOrder[2] := 1;
			arr_sint_StartOrder[3] := 2;
		ELSE
			arr_sint_StartOrder[2] := 2;
			arr_sint_StartOrder[3] := 1;
		END_IF
	END_IF
	arr_real_Steps[1]	:= real_Size_Step1_kW;
	arr_real_Steps[2]	:= real_Size_Step2_kW;
	arr_real_Steps[3]	:= real_Size_Step3_kW;
	
	arr_real_LoadSize[1] :=   arr_real_Steps[arr_sint_StartOrder[1]];
	arr_real_LoadSize[2] :=   arr_real_Steps[arr_sint_StartOrder[2]];
	arr_real_LoadSize[3] :=   arr_real_Steps[arr_sint_StartOrder[3]];
	
END_IF



// hour counter for each step
fb_HourCounter_Step1(	mCounterON:= m_Step1, 
						realHours=> real_Hours_Step1);
						
fb_HourCounter_Step2(	mCounterON:= m_Step2, 
						realHours=> real_Hours_Step2);
						
fb_HourCounter_Step3(	mCounterON:= m_Step3, 
						realHours=> real_Hours_Step3);

END_FUNCTION_BLOCK

// ---- FB/FB_HourCounter.TcPOU
FUNCTION_BLOCK FB_HourCounter
VAR_INPUT
	mCounterON								: BOOL;
END_VAR
VAR_OUTPUT
	realHours								: REAL;
END_VAR
VAR
	wSecond_old: WORD;
	fbGetSystemTime							: NT_GetTime;																					//Function to read out the windows system time on the local plc
	timGetTime								: TON;																							//Timer to activate the function tho read out the windows system time
END_VAR
VAR PERSISTENT
	udintEngineRunningSeconds				: UDINT;
	realHours_Persistent					: REAL;
END_VAR

IF mCounterON THEN
	IF fbGetSystemTime.TIMESTR.wSecond<>wSecond_old THEN
		udintEngineRunningSeconds:=udintEngineRunningSeconds+1;
	END_IF
END_IF
wSecond_old:=fbGetSystemTime.TIMESTR.wSecond;
realHours:=UDINT_TO_REAL(udintEngineRunningSeconds)/3600;
realHours_Persistent:=realHours;

timGetTime(IN:= NOT timGetTime.Q, PT:= T#1S, Q=> , ET=> );

fbGetSystemTime(
	NETID:= , 
	START:= timGetTime.Q AND NOT fbGetSystemTime.BUSY, 
	TMOUT:= , 
	BUSY=> , 
	ERR=> , 
	ERRID=> , 
	TIMESTR=> );

END_FUNCTION_BLOCK

// ---- POUs/prgPersistent.TcPOU
PROGRAM prgPersistent
VAR
	fbUSV		: FB_WritePersistentData_CX81xx;
	fb_Reboot		: NT_reboot;
	m_Reboot		: BOOL:=FALSE;
	uinit_KbusState: UINT;						//{#lynus.ag#()}
END_VAR

fbUSV(
	eSaveModeData:= eUSVSaveMode.eSaveWhenPowerfail, 
	bLoadPersistentDataOk=> , 
	bPowerFailDetect=> , 
	bError=> , 
	bySaveProcess=> , 
	dwStorageLast24h=> , 
	udiErrorCode=> );
	
	
fb_Reboot(	netid := '',
			delay := 2,
			start := m_Reboot);
	


uinit_KbusState := prgGrid.fbKBusState.uiKBusState_OUT;

END_PROGRAM

// ---- FB/FB_RAMP.TcPOU
FUNCTION_BLOCK FB_RAMP
VAR_INPUT
	realRampInput: REAL;		(* input value *)
	mEnableRamp: BOOL;			(* bit=0:Output=Input, bit=1: Ramp active, mZeroOutout has higher priority *)
	mZeroOutput:BOOL;			(* bit=0 normal operation, bit=1 output zero *)
	realRampSpeed: REAL;		(* speed value/second *)
	realRampSampleTime: REAL; 	(* based on 100ns increments *)
	realEqualize: REAL;
END_VAR
VAR_OUTPUT
	realRampOutput: REAL;		(* output value *)
	mRampSaturised: BOOL;		(* ramp on the end *)
END_VAR

VAR
END_VAR

(* 	24NOV2010:
	- new input variable: equalize value => when intput - output < equalize vale then output = input
*)
IF mEnableRamp AND NOT mZeroOutput THEN
	IF ABS(realRampOutput-realRampInput)<realEqualize THEN
		realRampOutput:=realRampInput; (* direct *)
		mRampSaturised:=TRUE;
	ELSE
		IF realRampOutput<realRampInput THEN (* increment *)
			realRampOutput:=realRampOutput+realRampSpeed*realRampSampleTime; (* realSampleTime in s *)
		END_IF
		IF realRampOutput>realRampInput THEN (* decrement *)
			realRampOutput:=realRampOutput-realRampSpeed*realRampSampleTime; (* realSampleTime in s *)
		END_IF
		mRampSaturised:=FALSE;
	END_IF
ELSE
	IF mZeroOutput THEN
		realRampOutput:=0;
	ELSE
		realRampOutput:=realRampInput; (* direct *)
	END_IF
END_IF

END_FUNCTION_BLOCK

// ---- FB/FB_Symo_PV_Inverter_FLOAT_1_DM_30_InclDisable_original.TcPOU
FUNCTION_BLOCK FB_Symo_PV_Inverter_FLOAT_1_DM_30_InclDisable_original
VAR_INPUT PERSISTENT
	bEnable						: BOOL;												//True = Function is enabled, FALSE = Function is dissabled, no new Data
	sIPAdress					: STRING(15);										//IP Adress from the Inverter
	arrUnitID_Inverter			: ARRAY[1..30] OF BYTE;								//Array with the Unit ID's from each Inverter (Max 30 Inverters) (ID = 1 to 247) (0 = No Inverter)
	arr_b_EnableWrite			: ARRAY[1..30] OF BOOL;								// Enable write function
	arr_m_DisableInverter		: ARRAY[1..30] OF BOOL;								// disable inverter 
	arr_int_InverterSetpoint	: ARRAY[1..30] OF INT;								// inverter setpoint i[1/100 %] 
END_VAR
VAR_OUTPUT
	arrDataSymo10				: ARRAY[1..30] OF ST_Symo_PV_OutData;				//Output structure with Data from Symo 10
	stDataEMPower_PV			: ST_ElectricMeter_Output_Power;					//Output structure with Data from Electric Meter PV (Power Data)
	stDataEMCounter_PV			: ST_ElectricMeter_Output_Counter;					//Output structure with Data from Electric Meter PV (Counter Data)
	diNrOfEM_OUT_PV				: DINT;												//Active Number from the Electric Meter for using on other functions
END_VAR
VAR
	fbElMeter					: FB_ElectricMeter;									//Electric Meter Function 
	fbNumberDevice				: FB_NumberOfDevice;								//Function block to calcualte the number of the Device
	fbConvertEnergyRegister		: FB_CV_WORD_TO_DWORD;								//Convert function
	fbMBRead_FC3				: FB_MBReadRegs;									//Modbus Read Function (FC3)
	fbMBWrite_FC16				: FB_MBWriteRegs;									//Modbus Write Function (FC16)
	timDelay					: TON;												//Timer for Delay between Requests
	timTimeout					: TON;												//Timer for Timeout
	timDissableFunctions		: TON;												//Timer to dissable the Function after Lynus_Standards.Constants_General.tTimeDissableLynusFunctions Days without connection to the Lynus Cloud
	timResetConnectionOnGVL		: TON;												//Timer to try reset the connection Flag on the GVL. (When somebody delete the Connection Function and make only a onlinechange)
	FPEnable					: R_TRIG;											//Internal positive Edge
	FPError_FC_3				: R_TRIG;											//Internal positive Edge
	FPError_FC_16				: R_TRIG;											//Internal positive Edge
	PD_String					: FB_PersistentData_String;							//Function to save persistent data 
	stFloat						: ST_UN_FLOAT_CONVERT_DWORD_REAL;					//Convert the Float Raw Value
	arrBuffer_FC3				: ARRAY[1..47] OF WORD;								//Buffer with Data from FC3
	arrBuffer_FC16				: ARRAY[1..6] OF WORD;								//Buffer with Data from FC16
	arrBuffer_FC16_old			: ARRAY[1..30,1..6] OF WORD;								//Buffer with Data from FC16
	arrUnitID_Inverter_CP		: ARRAY[1..30] OF BYTE;								//Array with unit IDs to compare it when we have a change on the Inputs
	arrCurrentL1				: ARRAY[1..30] OF LREAL;							//Array with the Current from L1 from each Inverter
	arrCurrentL2				: ARRAY[1..30] OF LREAL;							//Array with the Current from L2 from each Inverter
	arrCurrentL3				: ARRAY[1..30] OF LREAL;							//Array with the Current from L3 from each Inverter
	arrVoltageL1L2				: ARRAY[1..30] OF LREAL;							//Array with the Voltage from L1-L2 from each Inverter
	arrVoltageL2L3				: ARRAY[1..30] OF LREAL;							//Array with the Voltage from L2-L3 from each Inverter
	arrVoltageL3L1				: ARRAY[1..30] OF LREAL;							//Array with the Voltage from L3-L1 from each Inverter
	arrVoltageL1N				: ARRAY[1..30] OF LREAL;							//Array with the Voltage from L1-N from each Inverter
	arrVoltageL2N				: ARRAY[1..30] OF LREAL;							//Array with the Voltage from L2-N from each Inverter
	arrVoltageL3N				: ARRAY[1..30] OF LREAL;							//Array with the Voltage from L3-N from each Inverter
	arrACPower					: ARRAY[1..30] OF LREAL;							//Array with the AC Power from each Inverter
	arrFrequency				: ARRAY[1..30] OF LREAL;							//Array with the Frequency from each Inverter
	arrApparentPower			: ARRAY[1..30] OF LREAL;							//Array with the Apparent Power from each Inverter
	arrReactivePower			: ARRAY[1..30] OF LREAL;							//Array with the Reactive Power from each Inverter
	arrProductionEnergy			: ARRAY[1..30] OF LREAL;							//Array with the Production Energy from each Inverter
	arrPD						: ARRAY[1..31] OF FB_PersistentData_Number;			//Function to save persistent data
	bErrorDevice				: BOOL;												//When 1 or more Inverters has a Error, then thsi Flag is true
	byInverterInProgress		: BYTE;												//Shows what Inverter is at the moment in Progress in the State machine to read out the data
	byTotalInverter				: BYTE;												//Summ of total Inverters. (Depends on the unit IDs that are not 0.) 
	byLPForInverter				: BYTE; 											//Variable for Loop to calculate some things for the Inverters
	byWaitInStep				: BYTE;												//Wait in Step before start to clean data on PLC
	iStateGVLData				: INT;												//State machine to handle the data on the GVL
	iStateModbusRead			: INT;												//State variable for Statemachine
	iStateModbusWrite			: INT;												//State variable for Statemachine
	iStateModbus_CP				: INT;												//Compare State variable
	diCounterForGVL				: DINT;												//Counter to clean old data on GVL
	lrCheckValue				: LREAL;											//Internal Value to check the value before convert
	lrCounterEnergyProduction	: LREAL;											//Check counter state before write new one
	iStateModbusError			: INT;											//State variable for Statemachine
	byInverterInProgressWrite	: BYTE;
	ton_Wait_write: Ton;
	x: WORD;
	int_WriteSucessCounter: INT;
END_VAR

// {attribute 'hide_all_locals'}

//Creator : Kai Ebensperger
//Company : Lynus AG
//Date : 28.04.2021
//Version : 1.0.0.0

//With this function its possible to read out values from the Symo 10 PV Inverter from the factory Fronius
//This Function read out the Values from 1 Fronius Datamanager with maximal 30 Inverter.
//The protocol to the Inverter is Modbus TCP
//Versions that are supported : 1.1.5-0
//Attention. To access the registers, an offset of 1 must always be subtracted. Register 40001 would then be on register 40000.
//This Function use the FLOAT Format
//You can query the register data of the individual devices using the Modbus device ID (UnitID).
//Each inverter has its own number stored on the display under "Setup" -> "Datcom"-> "Inverter number".
//Inverter number 00 = Modbus ID 100
//Inverter number 01 = Modbus ID 01
//Inverter number 02 = Modbus ID 02 etc.
//Internal in the GVL this function is 1 PV Plant. We display the summ ov all values from each Inverter

//Changes about AC power
//Date : 29.03.2020
//Version : 1.1.0.0

//Date : 22.12.2022
//Version : 1.2.0.0
// STEFAN: added write to setpoint to inverter


//NOTE for diNr.....Designation => 
//_IN = Here Data come in from other Functions or go out to other functions about the GVL
//_OUT = Here Data go out to other functions about the GVL

(*------------------------------------------------------------------------------------------General Input Part---------------------------------------------------------------------------------------------*)

//Check limitation
FOR byLPForInverter := 1 TO 30 BY 1 DO
	arrUnitID_Inverter[byLPForInverter] := LIMIT(0,arrUnitID_Inverter[byLPForInverter],247);
END_FOR

(*-------------------------------------------------------------Calcualte the number of EM System---------------------------------------------------------------*)

fbNumberDevice(
	diActualNumberOfDevices:= Lynus_Standards.GVL_Energy.stNumberOfDevices.diNumberOfElectricMeters, 
	diMaxNumberOfDevices:= Constants_Energy.diMaxNumberOfElectricMeters, 
	udiCounterOnlineChange:= TwinCAT_SystemInfoVarList._AppInfo.OnlineChangeCnt, 
	bNumberIsCalculatet=> , 
	bFPNumberIsCalculatet=> , 
	bOnlineChange=> , 
	diNumberForThisDevice=> diNrOfEM_OUT_PV, 
	diNumberOfTotalDevices=> );

//Write new Numer on GVL
IF fbNumberDevice.bFPNumberIsCalculatet THEN
	Lynus_Standards.GVL_Energy.stNumberOfDevices.diNumberOfElectricMeters := fbNumberDevice.diNumberOfTotalDevices;	
END_IF 

//Delete old Number on GVL
IF fbNumberDevice.bOnlineChange THEN 
	Lynus_Standards.GVL_Energy.stNumberOfDevices.diNumberOfElectricMeters := diNrOfEM_OUT_PV;	
		iStateGVLData := 1; 
END_IF

(*-------------------------------------------------------------Service from Backend is ready and check the connection to backen for dissabel/enable Function---------------------------------------------------------------*)

//Try to reset the variable for connection on the GVL. When all is normal then the Lynus Mqtt connection function set this variable to true in the next cycle
//When we have no connection to the backend then after Lynus_Standards.Constants_General.tTimeDissableLynusFunctions days the Function is dissabled with all of his functionalities
timResetConnectionOnGVL(IN:= NOT timResetConnectionOnGVL.Q, PT:= T#1H, Q=> , ET=> );
	IF timResetConnectionOnGVL.Q THEN Lynus_Standards.GVL_Communicator.bStateConnectionToEnableFunctions := FALSE; END_IF
		IF NOT Lynus_Standards.GVL_Communicator.bStateConnectionToEnableFunctions THEN timDissableFunctions.IN := TRUE; ELSE timDissableFunctions.IN := FALSE; END_IF  
			timDissableFunctions(IN:= , PT:= Lynus_Standards.Constants_General.tTimeDissableLynusFunctions, Q=> , ET=> );

(*------------------------------------------------------------------------------------------Calcualte the Max Number of Inverters---------------------------------------------------------------------------------------------*)
	
byTotalInverter := 0;
	FOR byLPForInverter := 1 TO 30 BY 1 DO
		IF arrUnitID_Inverter[byLPForInverter] <> 0 THEN byTotalInverter := byTotalInverter + 1; END_IF 
	END_FOR	
	
(*------------------------------------------------------------------------------------------State Machine---------------------------------------------------------------------------------------------*)
	
//Enable
FPEnable(CLK:= bEnable, Q=> );
	IF FPEnable.Q AND iStateModbusRead = 0 AND byTotalInverter > 0 THEN iStateModbusRead := 1; END_IF
		IF NOT bEnable OR timDissableFunctions.Q OR byTotalInverter = 0 OR MEMCMP(ADR(arrUnitID_Inverter),ADR(arrUnitID_Inverter_CP),SIZEOF(arrUnitID_Inverter_CP)) <> 0 THEN iStateModbusRead := 0; END_IF

//Timer for delay
timDelay(IN:= , PT:= T#50MS, Q=> , ET=> );	

//Timer for Timeout in Statemachine
	IF iStateModbusRead = iStateModbus_CP THEN timTimeout.IN := TRUE; ELSE timTimeout.IN := FALSE; END_IF
		IF iStateModbusRead = 0 THEN timTimeout.IN := FALSE; END_IF
timTimeout(IN:= , PT:= T#20S, Q=> , ET=> );	

//Statemachine
CASE iStateModbusRead OF
	
	0://Init Step
		iStateModbus_CP := iStateModbusRead;
			timDelay.IN := FALSE;
		
		FOR byLPForInverter := 1 TO 30 BY 1 DO 
			arrDataSymo10[byLPForInverter].bFunctionIsActive := FALSE;
				arrDataSymo10[byLPForInverter].eOperatingStateInverter := E_Symo_PV_OperatingState.eNoDataReceived;
					arrDataSymo10[byLPForInverter].lrPowerAcInverter := 0;
			arrCurrentL1[byLPForInverter] := 0;
				arrCurrentL2[byLPForInverter] := 0;
			arrCurrentL3[byLPForInverter] := 0;
				arrVoltageL1L2[byLPForInverter] := 0;
			arrVoltageL2L3[byLPForInverter] := 0;
				arrVoltageL3L1[byLPForInverter] := 0;
			arrVoltageL1N[byLPForInverter] := 0;
				arrVoltageL2N[byLPForInverter] := 0;
			arrVoltageL3N[byLPForInverter] := 0;
				arrACPower[byLPForInverter] := 0;
			arrFrequency[byLPForInverter] := 0;
				arrApparentPower[byLPForInverter] := 0;
			arrReactivePower[byLPForInverter] := 0;
				arrProductionEnergy[byLPForInverter] := 0;
		END_FOR
				fbMBRead_FC3.bExecute := FALSE;
					lrCheckValue := 0;
			
		//After reset the Arrays when we have a change on the Unit ID's we restart the State Machine
		IF MEMCMP(ADR(arrUnitID_Inverter),ADR(arrUnitID_Inverter_CP),SIZEOF(arrUnitID_Inverter_CP)) <> 0 AND bEnable AND byTotalInverter > 0 THEN
			iStateModbusRead := 1;
				arrUnitID_Inverter_CP := arrUnitID_Inverter;
		END_IF
		
	1://Search the Unit ID to read out the Data for each Inverter with Unit ID <> 0
		iStateModbus_CP := iStateModbusRead;
		
		IF byInverterInProgress >= 30 THEN byInverterInProgress := 0; END_IF
		
		byInverterInProgress := byInverterInProgress + 1;
			byInverterInProgress := LIMIT(1,byInverterInProgress,30);	
		
		IF arrUnitID_Inverter[byInverterInProgress] <> 0 THEN iStateModbusRead := 2; END_IF
				
	2://Read out first Registers from 40072 to 40118
		arrDataSymo10[byInverterInProgress].bFunctionIsActive := TRUE;
			iStateModbus_CP := iStateModbusRead;
		
		fbMBRead_FC3.nQuantity := 47;
			fbMBRead_FC3.nMBAddr := 40071;
				fbMBRead_FC3.bExecute := TRUE;
					fbMBRead_FC3.nUnitID := arrUnitID_Inverter[byInverterInProgress];
			
		IF fbMBRead_FC3.bBusy THEN timDelay.IN := TRUE; END_IF
		
		//Wait for Delay, copy Data and then next step
		IF NOT fbMBRead_FC3.bBusy AND NOT fbMBRead_FC3.bError AND timDelay.Q THEN
			//Copy Data Current L1
			fbConvertEnergyRegister(wInputValue_1:= arrBuffer_FC3[3], wInputValue_2:= arrBuffer_FC3[4], eByteOrderForConvert:= eByteOrder.eBigEndian, dwOutputValue=> );
				stFloat.dwRawValue := fbConvertEnergyRegister.dwOutputValue;
					lrCheckValue := stFloat.rValueFloat;	
						IF lrCheckValue >= - 3.402823E+38 AND lrCheckValue <= 3.402823E+38 THEN 
							arrCurrentL1[byInverterInProgress] := lrCheckValue;
						ELSE
							iStateModbusRead := 300;
								arrDataSymo10[byInverterInProgress].eErrorState := E_Symo_PV_Error.eSymo10TooBigValueReceived;		
						END_IF
			//Copy Data Current L2
			fbConvertEnergyRegister(wInputValue_1:= arrBuffer_FC3[5], wInputValue_2:= arrBuffer_FC3[6], eByteOrderForConvert:= eByteOrder.eBigEndian, dwOutputValue=> );
				stFloat.dwRawValue := fbConvertEnergyRegister.dwOutputValue;
					lrCheckValue := stFloat.rValueFloat;	
						IF lrCheckValue >= - 3.402823E+38 AND lrCheckValue <= 3.402823E+38 THEN 
							arrCurrentL2[byInverterInProgress] := lrCheckValue;
						ELSE
							iStateModbusRead := 300;
								arrDataSymo10[byInverterInProgress].eErrorState := E_Symo_PV_Error.eSymo10TooBigValueReceived;		
						END_IF
			//Copy Data Current L3
			fbConvertEnergyRegister(wInputValue_1:= arrBuffer_FC3[7], wInputValue_2:= arrBuffer_FC3[8], eByteOrderForConvert:= eByteOrder.eBigEndian, dwOutputValue=> );
				stFloat.dwRawValue := fbConvertEnergyRegister.dwOutputValue;
					lrCheckValue := stFloat.rValueFloat;	
						IF lrCheckValue >= - 3.402823E+38 AND lrCheckValue <= 3.402823E+38 THEN 
							arrCurrentL3[byInverterInProgress] := lrCheckValue;
						ELSE
							iStateModbusRead := 300;
								arrDataSymo10[byInverterInProgress].eErrorState := E_Symo_PV_Error.eSymo10TooBigValueReceived;		
						END_IF
			//Copy Data Voltage L1-L2
			fbConvertEnergyRegister(wInputValue_1:= arrBuffer_FC3[9], wInputValue_2:= arrBuffer_FC3[10], eByteOrderForConvert:= eByteOrder.eBigEndian, dwOutputValue=> );
				stFloat.dwRawValue := fbConvertEnergyRegister.dwOutputValue;
					lrCheckValue := stFloat.rValueFloat;	
						IF lrCheckValue >= - 3.402823E+38 AND lrCheckValue <= 3.402823E+38 THEN 
							arrVoltageL1L2[byInverterInProgress] := lrCheckValue;
						ELSE
							iStateModbusRead := 300;
								arrDataSymo10[byInverterInProgress].eErrorState := E_Symo_PV_Error.eSymo10TooBigValueReceived;		
						END_IF
			//Copy Data Voltage L2-L3
			fbConvertEnergyRegister(wInputValue_1:= arrBuffer_FC3[11], wInputValue_2:= arrBuffer_FC3[12], eByteOrderForConvert:= eByteOrder.eBigEndian, dwOutputValue=> );
				stFloat.dwRawValue := fbConvertEnergyRegister.dwOutputValue;
					lrCheckValue := stFloat.rValueFloat;	
						IF lrCheckValue >= - 3.402823E+38 AND lrCheckValue <= 3.402823E+38 THEN 
							arrVoltageL2L3[byInverterInProgress] := lrCheckValue;
						ELSE
							iStateModbusRead := 300;
								arrDataSymo10[byInverterInProgress].eErrorState := E_Symo_PV_Error.eSymo10TooBigValueReceived;		
						END_IF
			//Copy Data Voltage L3-L1
			fbConvertEnergyRegister(wInputValue_1:= arrBuffer_FC3[13], wInputValue_2:= arrBuffer_FC3[14], eByteOrderForConvert:= eByteOrder.eBigEndian, dwOutputValue=> );
				stFloat.dwRawValue := fbConvertEnergyRegister.dwOutputValue;
					lrCheckValue := stFloat.rValueFloat;	
						IF lrCheckValue >= - 3.402823E+38 AND lrCheckValue <= 3.402823E+38 THEN 
							arrVoltageL3L1[byInverterInProgress] := lrCheckValue;
						ELSE
							iStateModbusRead := 300;
								arrDataSymo10[byInverterInProgress].eErrorState := E_Symo_PV_Error.eSymo10TooBigValueReceived;		
						END_IF
			//Copy Data Voltage L1-N
			fbConvertEnergyRegister(wInputValue_1:= arrBuffer_FC3[15], wInputValue_2:= arrBuffer_FC3[16], eByteOrderForConvert:= eByteOrder.eBigEndian, dwOutputValue=> );
				stFloat.dwRawValue := fbConvertEnergyRegister.dwOutputValue;
					lrCheckValue := stFloat.rValueFloat;	
						IF lrCheckValue >= - 3.402823E+38 AND lrCheckValue <= 3.402823E+38 THEN 
							arrVoltageL1N[byInverterInProgress] := lrCheckValue;
						ELSE
							iStateModbusRead := 300;
								arrDataSymo10[byInverterInProgress].eErrorState := E_Symo_PV_Error.eSymo10TooBigValueReceived;		
						END_IF
			//Copy Data Voltage L2-N
			fbConvertEnergyRegister(wInputValue_1:= arrBuffer_FC3[17], wInputValue_2:= arrBuffer_FC3[18], eByteOrderForConvert:= eByteOrder.eBigEndian, dwOutputValue=> );
				stFloat.dwRawValue := fbConvertEnergyRegister.dwOutputValue;
					lrCheckValue := stFloat.rValueFloat;	
						IF lrCheckValue >= - 3.402823E+38 AND lrCheckValue <= 3.402823E+38 THEN 
							arrVoltageL2N[byInverterInProgress] := lrCheckValue;
						ELSE
							iStateModbusRead := 300;
								arrDataSymo10[byInverterInProgress].eErrorState := E_Symo_PV_Error.eSymo10TooBigValueReceived;		
						END_IF
			//Copy Data Voltage L3-N
			fbConvertEnergyRegister(wInputValue_1:= arrBuffer_FC3[19], wInputValue_2:= arrBuffer_FC3[20], eByteOrderForConvert:= eByteOrder.eBigEndian, dwOutputValue=> );
				stFloat.dwRawValue := fbConvertEnergyRegister.dwOutputValue;
					lrCheckValue := stFloat.rValueFloat;	
						IF lrCheckValue >= - 3.402823E+38 AND lrCheckValue <= 3.402823E+38 THEN 
							arrVoltageL3N[byInverterInProgress] := lrCheckValue;
						ELSE
							iStateModbusRead := 300;
								arrDataSymo10[byInverterInProgress].eErrorState := E_Symo_PV_Error.eSymo10TooBigValueReceived;		
						END_IF
			//Copy Data AC Power
			fbConvertEnergyRegister(wInputValue_1:= arrBuffer_FC3[21], wInputValue_2:= arrBuffer_FC3[22], eByteOrderForConvert:= eByteOrder.eBigEndian, dwOutputValue=> );
				stFloat.dwRawValue := fbConvertEnergyRegister.dwOutputValue;
					lrCheckValue := stFloat.rValueFloat;	
						IF lrCheckValue >= - 3.402823E+38 AND lrCheckValue <= 3.402823E+38 THEN 
							arrACPower[byInverterInProgress] := lrCheckValue;
								arrDataSymo10[byInverterInProgress].lrPowerAcInverter := arrACPower[byInverterInProgress] / 1000;
						ELSE
							iStateModbusRead := 300;
								arrDataSymo10[byInverterInProgress].eErrorState := E_Symo_PV_Error.eSymo10TooBigValueReceived;		
						END_IF
			//Copy Data Frequency
			fbConvertEnergyRegister(wInputValue_1:= arrBuffer_FC3[23], wInputValue_2:= arrBuffer_FC3[24], eByteOrderForConvert:= eByteOrder.eBigEndian, dwOutputValue=> );
				stFloat.dwRawValue := fbConvertEnergyRegister.dwOutputValue;
					lrCheckValue := stFloat.rValueFloat;	
						IF lrCheckValue >= - 3.402823E+38 AND lrCheckValue <= 3.402823E+38 THEN 
							arrFrequency[byInverterInProgress] := lrCheckValue;
						ELSE
							iStateModbusRead := 300;
								arrDataSymo10[byInverterInProgress].eErrorState := E_Symo_PV_Error.eSymo10TooBigValueReceived;		
						END_IF
			//Copy Data Apparent Power
			fbConvertEnergyRegister(wInputValue_1:= arrBuffer_FC3[25], wInputValue_2:= arrBuffer_FC3[26], eByteOrderForConvert:= eByteOrder.eBigEndian, dwOutputValue=> );
				stFloat.dwRawValue := fbConvertEnergyRegister.dwOutputValue;
					lrCheckValue := stFloat.rValueFloat;	
						IF lrCheckValue >= - 3.402823E+38 AND lrCheckValue <= 3.402823E+38 THEN 
							arrApparentPower[byInverterInProgress] := lrCheckValue;
						ELSE
							iStateModbusRead := 300;
								arrDataSymo10[byInverterInProgress].eErrorState := E_Symo_PV_Error.eSymo10TooBigValueReceived;		
						END_IF
			//Copy Data Reactive Power
			fbConvertEnergyRegister(wInputValue_1:= arrBuffer_FC3[27], wInputValue_2:= arrBuffer_FC3[28], eByteOrderForConvert:= eByteOrder.eBigEndian, dwOutputValue=> );
				stFloat.dwRawValue := fbConvertEnergyRegister.dwOutputValue;
					lrCheckValue := stFloat.rValueFloat;	
						IF lrCheckValue >= - 3.402823E+38 AND lrCheckValue <= 3.402823E+38 THEN 
							arrReactivePower[byInverterInProgress] := lrCheckValue;
						ELSE
							iStateModbusRead := 300;
								arrDataSymo10[byInverterInProgress].eErrorState := E_Symo_PV_Error.eSymo10TooBigValueReceived;		
						END_IF
			//Copy Data AC production Energy
			fbConvertEnergyRegister(wInputValue_1:= arrBuffer_FC3[31], wInputValue_2:= arrBuffer_FC3[32], eByteOrderForConvert:= eByteOrder.eBigEndian, dwOutputValue=> );
				stFloat.dwRawValue := fbConvertEnergyRegister.dwOutputValue;
					lrCheckValue := stFloat.rValueFloat;	
						IF lrCheckValue >= - 3.402823E+38 AND lrCheckValue <= 3.402823E+38 THEN 
							arrProductionEnergy[byInverterInProgress] := lrCheckValue / 1000;
						ELSE
							iStateModbusRead := 300;
								arrDataSymo10[byInverterInProgress].eErrorState := E_Symo_PV_Error.eSymo10TooBigValueReceived;		
						END_IF
			//Operating State		
			IF arrBuffer_FC3[47] = 1 THEN arrDataSymo10[byInverterInProgress].eOperatingStateInverter := E_Symo_PV_OperatingState.eOff;
				ELSIF arrBuffer_FC3[47] = 2 THEN arrDataSymo10[byInverterInProgress].eOperatingStateInverter := E_Symo_PV_OperatingState.eSleeping;
				ELSIF arrBuffer_FC3[47] = 3 THEN arrDataSymo10[byInverterInProgress].eOperatingStateInverter := E_Symo_PV_OperatingState.eStartingUp;
				ELSIF arrBuffer_FC3[47] = 4 THEN arrDataSymo10[byInverterInProgress].eOperatingStateInverter := E_Symo_PV_OperatingState.eTrackingPowerPoint;
				ELSIF arrBuffer_FC3[47] = 5 THEN arrDataSymo10[byInverterInProgress].eOperatingStateInverter := E_Symo_PV_OperatingState.eForcedPowerReduction;
				ELSIF arrBuffer_FC3[47] = 6 THEN arrDataSymo10[byInverterInProgress].eOperatingStateInverter := E_Symo_PV_OperatingState.eShuttingDown;
				ELSIF arrBuffer_FC3[47] = 7 THEN arrDataSymo10[byInverterInProgress].eOperatingStateInverter := E_Symo_PV_OperatingState.eFaults;
				ELSIF arrBuffer_FC3[47] = 8 THEN arrDataSymo10[byInverterInProgress].eOperatingStateInverter := E_Symo_PV_OperatingState.eStandby;
				ELSE arrDataSymo10[byInverterInProgress].eOperatingStateInverter := E_Symo_PV_OperatingState.eNoDataReceived;
			END_IF
			//Next Step
			IF iStateModbusRead = 2 THEN
				fbMBRead_FC3.bExecute := FALSE;
					timDelay.IN := FALSE;
						iStateModbusRead := 3;
							arrDataSymo10[byInverterInProgress].bError := FALSE; 
								arrDataSymo10[byInverterInProgress].eErrorState := E_Symo_PV_Error.eNoError;
			END_IF
		END_IF
			
		//Error from Inverter
		IF NOT fbMBRead_FC3.bBusy AND NOT fbMBRead_FC3.bError AND timDelay.Q AND arrDataSymo10[byInverterInProgress].eOperatingStateInverter = E_Symo_PV_OperatingState.eFaults THEN
			iStateModbusRead := 300;
				arrDataSymo10[byInverterInProgress].eErrorState := E_Symo_PV_Error.eSymo10Error;
		END_IF
	 
		//Error or Timeout
		IF FPError_FC_3.Q OR timTimeout.Q THEN
			iStateModbusRead := 300;
				arrDataSymo10[byInverterInProgress].eErrorState := E_Symo_PV_Error.eModbusTCPError;
		END_IF

	3://Calculate the sum of the values
		iStateModbus_CP := iStateModbusRead;
		
		lrCounterEnergyProduction := 0;
			fbElMeter.lrCurrentL1 := 0;
		fbElMeter.lrCurrentL2 := 0;	
			fbElMeter.lrCurrentL3 := 0;
		fbElMeter.lrVoltageL1N := 0;
			fbElMeter.lrVoltageL2N := 0;
		fbElMeter.lrVoltageL3N := 0;
			fbElMeter.lrVoltageL1L2 := 0;
		fbElMeter.lrVoltageL2L3 := 0;
			fbElMeter.lrVoltageL3L1 := 0;
		fbElMeter.lrPowerTotal := 0;
			fbElMeter.lrFrequency := 0;
		fbElMeter.lrReactivePowerTotal := 0;
			fbElMeter.lrApparentPowerTotal := 0;
		
		FOR byLPForInverter := 1 TO 30 BY 1 DO 
			lrCounterEnergyProduction := lrCounterEnergyProduction + arrProductionEnergy[byLPForInverter];
			IF lrCounterEnergyProduction > fbElMeter.lrCounterEnergyT1_Production THEN
				fbElMeter.lrCounterEnergyT1_Production := lrCounterEnergyProduction;
			END_IF
				fbElMeter.lrCurrentL1 := fbElMeter.lrCurrentL1 + arrCurrentL1[byLPForInverter];
			fbElMeter.lrCurrentL2 := fbElMeter.lrCurrentL2 + arrCurrentL2[byLPForInverter];	
				fbElMeter.lrCurrentL3 := fbElMeter.lrCurrentL3 + arrCurrentL3[byLPForInverter];
			IF byTotalInverter > 0 THEN
				fbElMeter.lrVoltageL1N := (fbElMeter.lrVoltageL1N + arrVoltageL1N[byLPForInverter]) / byTotalInverter;
					fbElMeter.lrVoltageL2N := (fbElMeter.lrVoltageL2N + arrVoltageL2N[byLPForInverter]) / byTotalInverter;
				fbElMeter.lrVoltageL3N := (fbElMeter.lrVoltageL3N + arrVoltageL3N[byLPForInverter]) / byTotalInverter;
					fbElMeter.lrVoltageL1L2 := (fbElMeter.lrVoltageL1L2 + arrVoltageL1L2[byLPForInverter]) / byTotalInverter;
				fbElMeter.lrVoltageL2L3 := (fbElMeter.lrVoltageL2L3 + arrVoltageL2L3[byLPForInverter]) / byTotalInverter;
					fbElMeter.lrVoltageL3L1 := (fbElMeter.lrVoltageL3L1 + arrVoltageL3L1[byLPForInverter]) / byTotalInverter;
				fbElMeter.lrFrequency := (fbElMeter.lrFrequency + arrFrequency[byLPForInverter]) / byTotalInverter;
			END_IF
					fbElMeter.lrPowerTotal := fbElMeter.lrPowerTotal + arrACPower[byLPForInverter];
				fbElMeter.lrReactivePowerTotal := fbElMeter.lrReactivePowerTotal + arrReactivePower[byLPForInverter];
					fbElMeter.lrApparentPowerTotal := fbElMeter.lrApparentPowerTotal + arrApparentPower[byLPForInverter];
		END_FOR	
					
		fbElMeter.lrTotalCounterEnergy_Production := fbElMeter.lrCounterEnergyT1_Production; 
		
			iStateModbusRead := 4;
	
	4://Wait and go to write
		iStateModbus_CP := iStateModbusRead;
		
		iStateModbusWrite := 1;
		iStateModbusRead := - 1;	
				
	300://Error
		iStateModbus_CP := iStateModbusRead;
		timDelay.IN := FALSE;
		fbMBRead_FC3.bExecute := FALSE;
		arrDataSymo10[byInverterInProgress].bError := TRUE;
		iStateModbusWrite := 1;
		iStateModbusRead := - 1;	
END_CASE
(*------------------------------------------------------------------------------------------State Machine Write---------------------------------------------------------------------------------------------*)	
	
CASE iStateModbusWrite OF	
	1://Search the Unit ID to read out the Data for each Inverter with Unit ID <> 0
		iStateModbus_CP := iStateModbusWrite;
		arr_int_InverterSetpoint[byInverterInProgressWrite] := LIMIT (0,arr_int_InverterSetpoint[byInverterInProgressWrite],10000);
		IF byInverterInProgressWrite >= 30 THEN byInverterInProgressWrite := 0; END_IF
		
		byInverterInProgressWrite := byInverterInProgressWrite + 1;
		byInverterInProgressWrite := LIMIT(1,byInverterInProgressWrite,30);	
		
		IF arrUnitID_Inverter[byInverterInProgressWrite] <> 0 THEN iStateModbusWrite := 2; END_IF
				

	2://write disable inverter bit
		iStateModbus_CP := iStateModbusWrite;	

		arrBuffer_FC16[1] := BOOL_TO_WORD(NOT arr_m_DisableInverter[byInverterInProgressWrite]);		// reg 40241 / sunspec 40242 Enumerated valued.  Connection control. 0: Disconnected 1: Connected
		arrBuffer_FC16[2] := INT_TO_WORD(arr_int_InverterSetpoint[byInverterInProgressWrite]);	// reg 40242 / sunspec 40243 Set power output to specified level. [1/100 %]
	//	arrBuffer_FC16[3] := ;																		// reg 40243 / sunspec 40244 Time window for power limit change. 0-300
	//	arrBuffer_FC16[4] := ;																		// reg 40244 / sunspec 40245 Timeout period for power limit. 0-28800
		arrBuffer_FC16[5] := 2;																		// reg 40245 / sunspec 40246 Ramp time for moving from current setpoint to new setpoint. 0 - 65534 (0xFFFF has the same effect as 0x0000)
		arrBuffer_FC16[6] := 1;																		// reg 40246 / sunspec 40247 Enumerated valued.  Throttle enable/disable control 0: Disabled 1: Enabled

		IF arr_b_EnableWrite[byInverterInProgressWrite] then 
				//AND (arrBuffer_FC16[1] <> arrBuffer_FC16_old[byInverterInProgressWrite,1] OR arrBuffer_FC16[2] <> arrBuffer_FC16_old[byInverterInProgressWrite,2]) THEN 
		
			fbMBWrite_FC16.nQuantity := 6;
			fbMBWrite_FC16.nMBAddr := 40241;
			fbMBWrite_FC16.nUnitID := arrUnitID_Inverter[byInverterInProgressWrite];
			fbMBWrite_FC16.bExecute := TRUE;
			
		 
				
			IF fbMBWrite_FC16.bBusy THEN timDelay.IN := TRUE; END_IF
		ELSE
			fbMBWrite_FC16.bExecute := FALSE;
			timDelay.IN := FALSE;
			// go to next write step
			iStateModbusWrite := 3;
		END_IF
	
		//Wait for Delay and then next step
		IF NOT fbMBWrite_FC16.bBusy AND NOT fbMBWrite_FC16.bError AND timDelay.Q THEN
			arrBuffer_FC16_old[byInverterInProgressWrite,1] := arrBuffer_FC16[1];
			arrBuffer_FC16_old[byInverterInProgressWrite,2] := arrBuffer_FC16[2];
			int_WriteSucessCounter :=int_WriteSucessCounter+1;
			
			fbMBWrite_FC16.bExecute := FALSE;
			timDelay.IN := FALSE;
			//Restart from new with the Read out part
			iStateModbusWrite := 3;
		END_IF
				
		//Error or Timout
		IF FPError_FC_16.Q OR timTimeout.Q THEN
			fbMBWrite_FC16.bExecute := FALSE;
			timDelay.IN := FALSE;
			iStateModbusError := 300;
		END_IF
	
	3:
		ton_Wait_write.IN:=TRUE;
		IF ton_Wait_write.Q THEN
			ton_Wait_write.IN:=FALSE;
			iStateModbusRead := 1;
			iStateModbusWrite := 0;
		END_IF
END_CASE

(*------------------------------------------------------------------------------------------State Machine Write---------------------------------------------------------------------------------------------*)	

CASE iStateModbusError OF
	
	300://Error
		iStateModbus_CP := iStateModbusError;
		timDelay.IN := FALSE;
		fbMBRead_FC3.bExecute := FALSE;
		fbMBWrite_FC16.bExecute := FALSE;
		arrDataSymo10[byInverterInProgressWrite].bError := TRUE;
		//Restart from new with the Read out part after an Error
		iStateModbusRead := 1;	
		iStateModbusError := 0;
		iStateModbusWrite := 0;
END_CASE
ton_Wait_write(pt:= T#2S);
(*------------------------------------------------------------------------------------------Modbus TCP Function---------------------------------------------------------------------------------------------*)

fbMBRead_FC3(	sIPAddr:= sIPAdress, 
				nTCPPort:= 502, 
				cbLength:= SIZEOF(arrBuffer_FC3), 
				pDestAddr:= ADR(arrBuffer_FC3), 
				tTimeout:= T#10S );
				
	FPError_FC_3(CLK:= fbMBRead_FC3.bError, Q=> );

fbMBWrite_FC16(
		sIPAddr		:= sIPAdress, 
		nTCPPort	:= 502, 
		cbLength	:= SIZEOF(arrBuffer_FC16), 
		pSrcAddr	:= ADR(arrBuffer_FC16),     
		tTimeout	:= T#10S );
		
FPError_FC_16(CLK:= fbMBWrite_FC16.bError, Q=> );
(*----------------------------------------------------------------------------------------Electric Meter Data----------------------------------------------------------------------------------------------*)

//Error and Warning
bErrorDevice := FALSE;
	FOR byLPForInverter := 1 TO 30 BY 1 DO
		IF arrDataSymo10[byLPForInverter].bError THEN bErrorDevice := TRUE; END_IF 
	END_FOR 

IF timDissableFunctions.Q THEN fbElMeter.bWarning := TRUE; fbElMeter.iWarningCode := 0; ELSE fbElMeter.bWarning := FALSE; END_IF   
	IF bErrorDevice OR Lynus_Standards.GVL_Energy.stNumberOfDevices.diNumberOfElectricMeters > Constants_Energy.diMaxNumberOfElectricMeters THEN fbElMeter.bError := TRUE; ELSE fbElMeter.bError := FALSE; END_IF  

IF Lynus_Standards.GVL_Energy.stNumberOfDevices.diNumberOfElectricMeters > Constants_Energy.diMaxNumberOfElectricMeters THEN fbElMeter.iErrorCode := 1;
ELSIF bErrorDevice THEN fbElMeter.iErrorCode := 0;
END_IF  

//Read Out Data done for EM Function
IF iStateModbusRead <> 3 THEN fbElMeter.bReadOutDataDone := TRUE; ELSE fbElMeter.bReadOutDataDone := FALSE; END_IF

//Function block for meter data
fbElMeter(
	bEnable:= bEnable AND NOT timDissableFunctions.Q, 
	bError:= , 
	bEnableReadOutFunction:= FALSE, 
	bWriteWithDelay:= TRUE,
	bPowerDataInvers:= TRUE, 
	bReadOutDataDone:= ,
	iTimeReadOutInterval:= , 
	iErrorCode:= , 
	iWarningCode:= , 
	lrTotalCounterEnergy_Consumption:= 0, 
	lrTotalCounterEnergy_Production:= , 
	lrCounterEnergyT1_Consumption:= 0, 
	lrCounterEnergyT2_Consumption:= 0, 
	lrCounterEnergyT1_Production:= , 
	lrCounterEnergyT2_Production:= 0, 
	lrCurrentL1:= , 
	lrVoltageL1N:= , 
	lrVoltageL1L2:= , 
	lrPowerL1:= 0, 
	lrCurrentL2:= , 
	lrVoltageL2N:= , 
	lrVoltageL2L3:= , 
	lrPowerL2:= 0, 
	lrCurrentL3:= , 
	lrVoltageL3N:= , 
	lrVoltageL3L1:= , 
	lrPowerL3:= 0, 
	lrPowerTotal:= , 
	lrFrequency:= , 
	lrReactivePowerTotal:= , 
	lrApparentPowerTotal:= , 
	tTimDelayOutput:= T#5S, 
	stDataEMOutPower=> , 
	stDataEMOutPowerDelay=> stDataEMPower_PV, 
	stDataEMOutCounter=> ,
	stDataEMOutCounterDelay=> stDataEMCounter_PV, 
	bReadOutMeter=> );

(*-----------------------------------------------------------Handle data to Global structure for the Electric Meter system-----------------------------------------------------------------*)

CASE iStateGVLData OF
	
	0://Init Step
		byWaitInStep := 0;
			diCounterForGVL := 1;
	
	1://Wait for 4 Steps before clean al Data on GVL
		byWaitInStep := byWaitInStep + 1;
			IF byWaitInStep >= 4 AND fbNumberDevice.bNumberIsCalculatet THEN iStateGVLData := 2; END_IF
				//To much Devices, back to the Init step
				IF byWaitInStep >= 4 AND NOT fbNumberDevice.bNumberIsCalculatet THEN iStateGVLData := 0; END_IF	
			
	2://Clear all Data in GVL
		Lynus_Standards.GVL_Energy.stDataElectricMeters[diCounterForGVL].bEnabled := FALSE;	
			Lynus_Standards.GVL_Energy.stDataElectricMeters[diCounterForGVL].byErrorWarning := 0;
				Lynus_Standards.GVL_Energy.stDataElectricMeters[diCounterForGVL].lrCounterEnergyT1_Consumption := 0;
					Lynus_Standards.GVL_Energy.stDataElectricMeters[diCounterForGVL].lrCounterEnergyT1_Production := 0;
						Lynus_Standards.GVL_Energy.stDataElectricMeters[diCounterForGVL].lrCounterEnergyT2_Consumption := 0;
							Lynus_Standards.GVL_Energy.stDataElectricMeters[diCounterForGVL].lrCounterEnergyT2_Production := 0;
								Lynus_Standards.GVL_Energy.stDataElectricMeters[diCounterForGVL].lrPower := 0;
									Lynus_Standards.GVL_Energy.stDataElectricMeters[diCounterForGVL].lrPowerConsumption := 0;
										Lynus_Standards.GVL_Energy.stDataElectricMeters[diCounterForGVL].lrPowerConsumption := 0;
											Lynus_Standards.GVL_Energy.stDataElectricMeters[diCounterForGVL].lrPowerProduction := 0;
												Lynus_Standards.GVL_Energy.stDataElectricMeters[diCounterForGVL].lrTotalCounterEnergy_Consumption := 0;
													Lynus_Standards.GVL_Energy.stDataElectricMeters[diCounterForGVL].lrTotalCounterEnergy_Production := 0;
		
		diCounterForGVL := diCounterForGVL + 1;
			diCounterForGVL := LIMIT(0,diCounterForGVL,Constants_Energy.diMaxNumberOfElectricMeters);
				//Back to the init step
				IF diCounterForGVL >= Constants_Energy.diMaxNumberOfElectricMeters THEN iStateGVLData := 0; END_IF

END_CASE 	 

IF diNrOfEM_OUT_PV > 0 AND fbNumberDevice.bNumberIsCalculatet THEN
	Lynus_Standards.GVL_Energy.stDataElectricMeters[diNrOfEM_OUT_PV].bEnabled := fbElMeter.stDataEMOutPower.bEnabled;
		Lynus_Standards.GVL_Energy.stDataElectricMeters[diNrOfEM_OUT_PV].byErrorWarning := fbElMeter.stDataEMOutPower.byErrorWarning;
			Lynus_Standards.GVL_Energy.stDataElectricMeters[diNrOfEM_OUT_PV].lrCounterEnergyT1_Consumption := fbElMeter.stDataEMOutCounter.lrCounterEnergyT1_Consumption;
				Lynus_Standards.GVL_Energy.stDataElectricMeters[diNrOfEM_OUT_PV].lrCounterEnergyT1_Production := fbElMeter.stDataEMOutCounter.lrCounterEnergyT1_Production;
					Lynus_Standards.GVL_Energy.stDataElectricMeters[diNrOfEM_OUT_PV].lrCounterEnergyT2_Consumption := fbElMeter.stDataEMOutCounter.lrCounterEnergyT2_Consumption;
						Lynus_Standards.GVL_Energy.stDataElectricMeters[diNrOfEM_OUT_PV].lrCounterEnergyT2_Production := fbElMeter.stDataEMOutCounter.lrCounterEnergyT2_Production;		
							Lynus_Standards.GVL_Energy.stDataElectricMeters[diNrOfEM_OUT_PV].lrPower := fbElMeter.stDataEMOutPower.lrPowerTotal;
								Lynus_Standards.GVL_Energy.stDataElectricMeters[diNrOfEM_OUT_PV].lrPowerConsumption := fbElMeter.stDataEMOutPower.lrPowerConsumption;
									Lynus_Standards.GVL_Energy.stDataElectricMeters[diNrOfEM_OUT_PV].lrPowerProduction := fbElMeter.stDataEMOutPower.lrPowerProduction;
										Lynus_Standards.GVL_Energy.stDataElectricMeters[diNrOfEM_OUT_PV].lrTotalCounterEnergy_Consumption := fbElMeter.stDataEMOutCounter.lrTotalCounterEnergy_Consumption;
											Lynus_Standards.GVL_Energy.stDataElectricMeters[diNrOfEM_OUT_PV].lrTotalCounterEnergy_Production := fbElMeter.stDataEMOutCounter.lrTotalCounterEnergy_Production;
END_IF

(*----------------------------------------------------------Save persistent data----------------------------------------------------------------*)

arrPD[1](lrValue:= BOOL_TO_LREAL(bEnable), bEventBasedActive=> );
arrPD[2](lrValue:= BYTE_TO_LREAL(arrUnitID_Inverter[1]), bEventBasedActive=> );
arrPD[3](lrValue:= BYTE_TO_LREAL(arrUnitID_Inverter[2]), bEventBasedActive=> );
arrPD[4](lrValue:= BYTE_TO_LREAL(arrUnitID_Inverter[3]), bEventBasedActive=> );
arrPD[5](lrValue:= BYTE_TO_LREAL(arrUnitID_Inverter[4]), bEventBasedActive=> );
arrPD[6](lrValue:= BYTE_TO_LREAL(arrUnitID_Inverter[5]), bEventBasedActive=> );
arrPD[7](lrValue:= BYTE_TO_LREAL(arrUnitID_Inverter[6]), bEventBasedActive=> );
arrPD[8](lrValue:= BYTE_TO_LREAL(arrUnitID_Inverter[7]), bEventBasedActive=> );
arrPD[9](lrValue:= BYTE_TO_LREAL(arrUnitID_Inverter[8]), bEventBasedActive=> );
arrPD[10](lrValue:= BYTE_TO_LREAL(arrUnitID_Inverter[9]), bEventBasedActive=> );
arrPD[11](lrValue:= BYTE_TO_LREAL(arrUnitID_Inverter[10]), bEventBasedActive=> );
arrPD[12](lrValue:= BYTE_TO_LREAL(arrUnitID_Inverter[11]), bEventBasedActive=> );
arrPD[13](lrValue:= BYTE_TO_LREAL(arrUnitID_Inverter[12]), bEventBasedActive=> );
arrPD[14](lrValue:= BYTE_TO_LREAL(arrUnitID_Inverter[13]), bEventBasedActive=> );
arrPD[15](lrValue:= BYTE_TO_LREAL(arrUnitID_Inverter[14]), bEventBasedActive=> );
arrPD[16](lrValue:= BYTE_TO_LREAL(arrUnitID_Inverter[15]), bEventBasedActive=> );
arrPD[17](lrValue:= BYTE_TO_LREAL(arrUnitID_Inverter[16]), bEventBasedActive=> );
arrPD[18](lrValue:= BYTE_TO_LREAL(arrUnitID_Inverter[17]), bEventBasedActive=> );
arrPD[19](lrValue:= BYTE_TO_LREAL(arrUnitID_Inverter[18]), bEventBasedActive=> );
arrPD[20](lrValue:= BYTE_TO_LREAL(arrUnitID_Inverter[19]), bEventBasedActive=> );
arrPD[21](lrValue:= BYTE_TO_LREAL(arrUnitID_Inverter[20]), bEventBasedActive=> );
arrPD[22](lrValue:= BYTE_TO_LREAL(arrUnitID_Inverter[21]), bEventBasedActive=> );
arrPD[23](lrValue:= BYTE_TO_LREAL(arrUnitID_Inverter[22]), bEventBasedActive=> );
arrPD[24](lrValue:= BYTE_TO_LREAL(arrUnitID_Inverter[23]), bEventBasedActive=> );
arrPD[25](lrValue:= BYTE_TO_LREAL(arrUnitID_Inverter[24]), bEventBasedActive=> );
arrPD[26](lrValue:= BYTE_TO_LREAL(arrUnitID_Inverter[25]), bEventBasedActive=> );
arrPD[27](lrValue:= BYTE_TO_LREAL(arrUnitID_Inverter[26]), bEventBasedActive=> );
arrPD[28](lrValue:= BYTE_TO_LREAL(arrUnitID_Inverter[27]), bEventBasedActive=> );
arrPD[29](lrValue:= BYTE_TO_LREAL(arrUnitID_Inverter[28]), bEventBasedActive=> );
arrPD[30](lrValue:= BYTE_TO_LREAL(arrUnitID_Inverter[29]), bEventBasedActive=> );
arrPD[31](lrValue:= BYTE_TO_LREAL(arrUnitID_Inverter[30]), bEventBasedActive=> );
PD_String(sText:= sIPAdress, bEventBasedActive=> );

END_FUNCTION_BLOCK
